ABB RobotStudio station: Project3.rsstnx

Station Project3 (saved by RobotStudio 25.5.11605.0)
Controller Robot, task T_ROB1: task frame (RAPID world) sits at (91.86, 0, 0) mm in the station
Controller Robot
  mechanical unit ROB_1: IRB1200_5_90_STD_03, 6 joints, base frame (0, 0, 0) mm
Layout (positions relative to the parent item):
  - IRB1200_5_90_STD_03 [mechanism, from %ABB.RobotStudio.Models.IRB1200%\IRB1200_5_90_STD_03.rslib] at (91.86, 0, 0) mm; joint values [0, 0.6721, 0.8136, 0, -0.9621, 0] (rad or m)
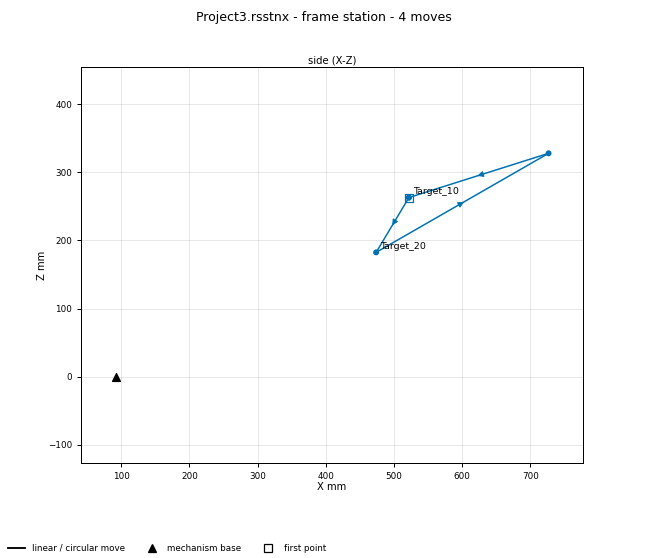
[picture p0: tool path of Project3.rsstnx in frame station, 4 of 4 moves have a stored position in this frame; points joined in program order, loops and branches not executed]
Targets, tools, work objects and paths stored in the station, written as RAPID:
! task T_ROB1
MODULE Module1
  CONST robtarget Target_10:=[[430.149444003,0,262.870109053],[0.50000002,0,0.866025392,0],[0,0,0,1],[9E+09,9E+09,9E+09,9E+09,9E+09,9E+09]];
  CONST robtarget Target_20:=[[382.118748209,0,182.513936698],[0.499999994,0,0.866025407,0],[0,0,0,1],[9E+09,9E+09,9E+09,9E+09,9E+09,9E+09]];
  CONST robtarget Target_30:=[[635.009450895,0,327.754464907],[0.50000002,0,0.866025392,0],[0,0,0,1],[9E+09,9E+09,9E+09,9E+09,9E+09,9E+09]];
  CONST robtarget Target_10_4:=[[430.149444003,0,262.870109053],[0.50000002,0,0.866025392,0],[0,0,0,1],[9E+09,9E+09,9E+09,9E+09,9E+09,9E+09]];
  PROC Path_10()
    MoveL Target_10,v1000,z100,tool0\WObj:=wobj0;
    MoveL Target_20,v1000,z100,tool0\WObj:=wobj0;
    SetDO out_1,1;
    WaitTime 1;
    MoveL Target_30,v1000,z100,tool0\WObj:=wobj0;
    WaitTime 1;
    SetDO out_1,0;
    WaitTime 1;
    MoveL Target_10_4,v1000,z100,tool0\WObj:=wobj0;
  ENDPROC
  PROC main()
    Path_10;
    SetDO out_0,1;
    WaitTime 0.5;
    SetDO out_0,0;
    WaitDI in_0,0;
  ENDPROC
ENDMODULE

